Omron CX-Programmer project NewProject (CX-Programmer 9.75)

# PLC OMRON: CP1E N30

## Global symbols (name address type ; comment)
C000 BOOL  ; C0

## Program NewProgram1 (cyclic task 0)
Local symbols
AirConditioner 100.06 BOOL  ; 100.06
Fan1 100.04 BOOL
Fan2 100.05 BOOL  ; 100.05
Lamp1 100.01 BOOL  ; 100.01
Lamp2 100.02 BOOL  ; 100.02
Lamp3 100.03 BOOL  ; 100.03
MainSupplly 100.00 BOOL  ; 100.00
Reset 0.04 BOOL  ; 0.04
Sensor 0.03 BOOL  ; 0.03
Sw1 0.00 BOOL  ; 0.00
Sw2 0.01 BOOL  ; 0.01
Sw3 0.02 BOOL  ; 0.02

### Section Section1

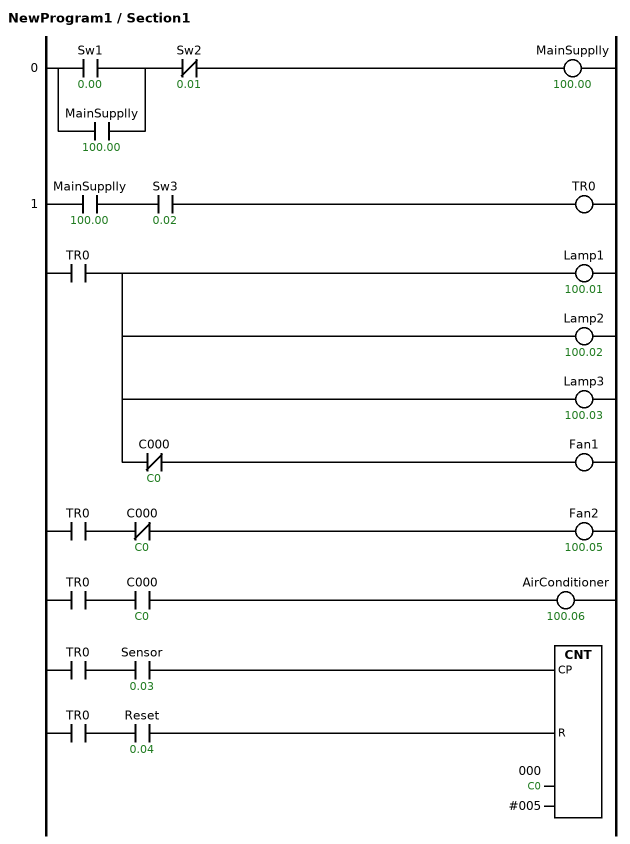
; rung 0
LD Sw1  ; 0.00
OR MainSupplly  ; 100.00
ANDNOT Sw2  ; 0.01
OUT MainSupplly  ; 100.00
; rung 1
LD MainSupplly  ; 100.00
AND Sw3  ; 0.02
OUT TR0
OUT Lamp1  ; 100.01
OUT Lamp2  ; 100.02
OUT Lamp3  ; 100.03
ANDNOT C000  ; C0
OUT Fan1
LD TR0
ANDNOT C000  ; C0
OUT Fan2  ; 100.05
LD TR0
AND C000  ; C0
OUT AirConditioner  ; 100.06
LD TR0
AND Sensor  ; 0.03
LD TR0
AND Reset  ; 0.04
CNT 000 #005  ; C0

### Section END
; rung 0
END(001)